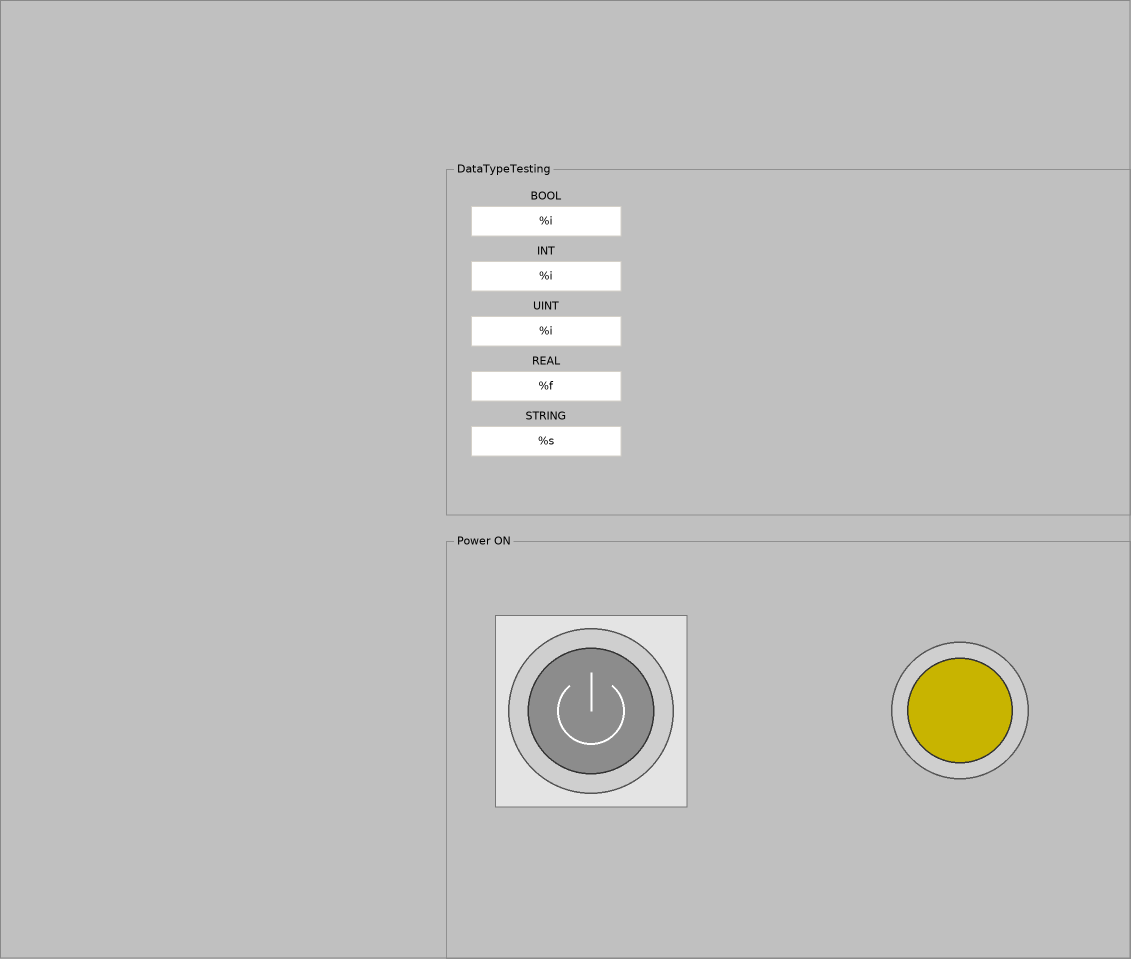
VISUALIZATION HMI  // 1131x959
    GroupBox (446,533 685x426), "Power ON"
        Lamp1 (434,90 160x175), variable: MAIN.bEnable, style: Lamp-Lamp1-Yellow
        PowerSwitch (49,63 192x230), variable: MAIN.bStart, behaviour: TOGGLE, style: Switch-PowerSwitch-Gray
    GroupBox (446,161 685x354), "DataTypeTesting"
        Textfield (25,45 150x30), "%i", text variable: MAIN.bEnable
        Textfield (25,100 150x30), "%i", text variable: MAIN.nINT
        Textfield (25,155 150x30), "%i", text variable: MAIN.nUINT
        Textfield (25,210 150x30), "%f", text variable: MAIN.fREAL
            OnMouseDown: write the text variable via Default
        Textfield (25,265 150x30), "%s", text variable: MAIN.sPowerStatus
            OnMouseDown: write the text variable via Default
        Label (25,20 150x30), "BOOL"
        Label (25,75 150x30), "INT"
        Label (25,130 150x30), "UINT"
        Label (25,185 150x30), "REAL"
        Label (25,240 150x30), "STRING"
END_VISUALIZATION

(* stored: Version 1.1.0.1, ProductVersion 3.1.4024.12
   Visu HMI: Id {dc07b08d-2694-4675-baa2-ef7f71b7e52d} *)
